{attribute 'TcGenerated'}
{attribute 'no-analysis'}
{attribute 'linkalways'}
// This function has been automatically generated from the project information.
VAR_GLOBAL CONSTANT
	{attribute 'const_non_replaced'}
	stLibVersion_FactoryIO_Library : ST_LibVersion := (iMajor := 0, iMinor := 0, iBuild := 7, iRevision := 0, nFlags := 0, sVersion := '0.0.7');
END_VAR

(* stored: Version 1.1.0.1
   GVL Global_Version: Id {c032101c-de01-4a2a-95b7-b05cac8199a8} *)
